FUNCTION_BLOCK ServoMotor IMPLEMENTS GpMotor
VAR_INPUT
END_VAR
VAR_OUTPUT
END_VAR
VAR
	driveControl1 : DriveControl; // Complex internal logic
		isRunning : BOOL:= FALSE ;
END_VAR


METHOD Start : BOOL
driveControl1.Enable();
driveControl1.MoveVelocity(3000);
isRunning := TRUE;
 Start := TRUE;
END_METHOD

METHOD Stop : BOOL
DriveCOntrol1.QuickStop();
isRunning := FALSE;
Stop := TRUE;
END_METHOD

END_FUNCTION_BLOCK

(* stored: Version 1.1.0.1, ProductVersion 3.1.4024.16
   POU ServoMotor: Id {3f3ec948-29f4-4471-ae7f-d0c24c896fb2}, SpecialFunc None
   Method Start: Id {5f1b2c96-eb69-475c-9549-f11631968d54}
   Method Stop: Id {bc7a5dc7-195b-4770-b908-e0c8473a5c21} *)
